VAR_GLOBAL
	instEmitter	:	FB_Emitter;	//Instanz Emitter 4m Rollenfoerderer
	CreateNewPart	:	BOOL;
END_VAR

(* stored: Version 1.1.0.1
   GVL Emitter: Id {6f5ea492-507e-4f6b-b498-dba00c51bd54} *)
